FUNCTION_BLOCK SNSVL_THMI (* HMI and Local Multicast elements for testing an instance of SNSVL. *)
  (* Standard: IEC 61499; Classification: HMI; ApplicationDomain: Process Control; Function: Test; Type: Sensor *)
  (* Version 0.0, 2006-08-02, JHC, Holobloc Inc *)
  (* Compiler header: package fb.rt.batch; import fb.rt.net.*; import fb.rt.hmi.*; import fb.rt.mva.FBMVCD; *)
  (* Compiler classdef: public class SNSVL_THMI extends FBMVCD *)
  (* Compiler Java Sun JDK 1.5.0 *)
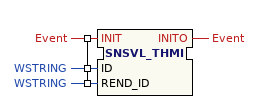
  EVENT_INPUT
    INIT WITH REND_ID, ID; (* Initialization Request *)
  END_EVENT
  EVENT_OUTPUT
    INITO; (* Initialization Confirm *)
  END_EVENT
  VAR_INPUT
    ID : WSTRING; (* Label for HMI elements, default = FB instance name *)
    REND_ID : WSTRING; (* Local Channel ID for rendering data *)
  END_VAR
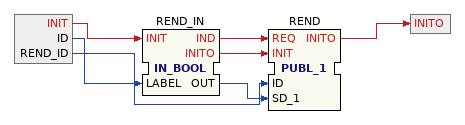
  FBS
    REND : PUBL_1;
    REND_IN : IN_BOOL;
  END_FBS
  EVENT_CONNECTIONS
    INIT TO REND_IN.INIT;
    REND_IN.IND TO REND.REQ;
    REND_IN.INITO TO REND.INIT;
    REND.INITO TO INITO;
  END_CONNECTIONS
  DATA_CONNECTIONS
    REND_ID TO REND.ID;
    ID TO REND_IN.LABEL;
    REND_IN.OUT TO REND.SD_1;
  END_CONNECTIONS
END_FUNCTION_BLOCK
